ABB RobotStudio station: ScenarioBrakeTest.rspag

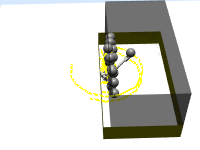
--- station ---
Station Solution10_1 (saved by RobotStudio 6.7.7850.130)
Controller IRB_6700_175kg_3.05m
  mechanical unit ROB_1: IRB6700_175_305__04, 6 joints, base frame (0, 0, 0) mm
Layout (positions relative to the parent item):
  - IRB6700_175_305__04 [mechanism, from Robots\IRB6700_175_305__04.rslib] at (0, 0, 0) mm; joint values [-1.1842, -1.1345, -1.3411, 0, 0.5236, 0] (rad or m)
  - MyNewTool [mechanism] at (-813.86, 1999.53, 2271.97) mm, rotated rx 0 ry -21.84 rz -67.85 deg
      TCP MyNewTool at (0, 0, 0) mm
      links: IsoPlate_large_sat
  - SafeSpaceGeometries [graphiccomponentgroup]
    - safety zone [part]
    - tcp blob [part] at (-813.86, 1999.53, 2271.97) mm, rotated rx 0 ry -21.84 rz -67.85 deg
    - tcp blob [part] at (-1295.95, 228.51, 2690.77) mm, rotated rx -180 ry 87.5 rz -10 deg
    - tcp blob [part] at (-2238.8, 394.76, 1689.63) mm, rotated rx -180 ry 50 rz -10 deg
    - tcp blob [part] at (2430.82, 428.62, 1082.75) mm, rotated rx 0 ry -62.5 rz -170 deg
    - tcp blob [part] at (2269.78, 400.22, 2021.28) mm, rotated rx 0 ry -31.25 rz -170 deg
    - tcp blob [part] at (1652.62, 291.4, 2738.82) mm, rotated rx 0 ry 0 rz -170 deg
    - tcp blob [part] at (758.42, 133.73, 3027.14) mm, rotated rx 0 ry 31.25 rz -170 deg
    - tcp blob [part] at (1942.58, 342.53, 1802.45) mm, rotated rx 0 ry -56.25 rz -170 deg
    - tcp blob [part] at (1681.88, 296.56, 2717.61) mm, rotated rx 0 ry -25 rz -170 deg
    - tcp blob [part] at (991.45, 174.82, 3362.65) mm, rotated rx 0 ry 6.25 rz -170 deg
    - tcp blob [part] at (863.06, 152.18, 2986.78) mm, rotated rx 0 ry -18.75 rz -170 deg
    - tcp blob [part] at (582.02, 504.32, 3027.14) mm, rotated rx 0 ry 31.25 rz -139.09 deg
    - tcp blob [part] at (82.99, 71.91, 2781.05) mm, rotated rx 0 ry -12.5 rz -139.09 deg
    - tcp blob [part] at (34.09, 103.78, 3551.67) mm, rotated rx 0 ry 12.5 rz -108.18 deg
    - tcp blob [part] at (34.26, 104.33, 2781.05) mm, rotated rx 0 ry -12.5 rz -108.18 deg
    - tcp blob [part] at (-24.07, 106.55, 3551.67) mm, rotated rx 0 ry 12.5 rz -77.27 deg
    - tcp blob [part] at (-24.19, 107.11, 2781.05) mm, rotated rx 0 ry -12.5 rz -77.27 deg
    - tcp blob [part] at (-531.44, 557.36, 3027.14) mm, rotated rx 0 ry 31.25 rz -46.36 deg
    - tcp blob [part] at (-75.78, 79.47, 2781.05) mm, rotated rx 0 ry -12.5 rz -46.36 deg
    - tcp blob [part] at (-1617.44, 447.17, 2738.82) mm, rotated rx 0 ry 0 rz -15.45 deg
    - tcp blob [part] at (-742.27, 205.22, 3027.14) mm, rotated rx 0 ry 31.25 rz -15.45 deg
    - tcp blob [part] at (-970.35, 268.27, 3362.65) mm, rotated rx 0 ry 6.25 rz -15.45 deg
    - tcp blob [part] at (-844.68, 233.53, 2986.78) mm, rotated rx 0 ry -18.75 rz -15.45 deg
    - tcp blob [part] at (1020.75, 282.21, 1205.4) mm, rotated rx -180 ry 55 rz -164.55 deg
    - tcp blob [part] at (1369.56, 378.64, 2484.63) mm, rotated rx -180 ry 80 rz -164.55 deg
    - tcp blob [part] at (1491.26, 412.29, 1540.36) mm, rotated rx -180 ry 48.75 rz -164.55 deg
    - tcp blob [part] at (1123.15, 310.52, 667.59) mm, rotated rx -180 ry 17.5 rz -164.55 deg
    - tcp blob [part] at (-1042.95, 183.9, 1205.4) mm, rotated rx -180 ry 55 rz -10 deg
    - tcp blob [part] at (-1399.35, 246.74, 2484.63) mm, rotated rx -180 ry 80 rz -10 deg
    - tcp blob [part] at (-1523.7, 268.67, 1540.36) mm, rotated rx -180 ry 48.75 rz -10 deg
    - tcp blob [part] at (-1147.59, 202.35, 667.59) mm, rotated rx -180 ry 17.5 rz -10 deg
    - tcp blob [part] at (-1669.17, 294.32, 3217.01) mm, rotated rx 0 ry 75 rz 170 deg
    - tcp blob [part] at (-2174.87, 383.49, 2414.57) mm, rotated rx -180 ry 73.75 rz -10 deg
    - tcp blob [part] at (-2197.25, 387.43, 1462.17) mm, rotated rx -180 ry 42.5 rz -10 deg
    - tcp blob [part] at (-1729.8, 305.01, 636.16) mm, rotated rx -180 ry 11.25 rz -10 deg
    - tcp blob [part] at (-1641.43, 289.43, 3240.22) mm, rotated rx 0 ry 50 rz 170 deg
    - tcp blob [part] at (-2433.72, 429.13, 2729.98) mm, rotated rx 0 ry 81.25 rz 170 deg
    - tcp blob [part] at (-2109.4, 371.94, 2506.76) mm, rotated rx 0 ry 56.25 rz 170 deg
    - fence_2000 [part]
    - fence_4000 [part]
    - fence_6000 [part]
  - Part_2 [part] at (-12128.6, -11086.49, -16.13) mm
Attachment: MyNewTool is attached to IRB6700_175_305__04 / Link6
Attachment: tcp blob is attached to IRB6700_175_305__04 / Link6
Collision set zone collisions: tcp blob against safety zone, near miss 0 m
Targets, tools, work objects and paths stored in the station and not in the controller backup, written as RAPID:
! task T_ROB1
MODULE Module1
  CONST robtarget Target_0112:=[[2430.822564059,428.619603359,1082.747931027],[0.074510479,-0.516799169,-0.045214069,-0.851658673],[-2,0,0,6],[9E+09,9E+09,9E+09,9E+09,9E+09,9E+09]];
  CONST robtarget Target_0113:=[[2430.822564059,428.619603359,1082.747931027],[0.074510479,-0.516799169,-0.045214069,-0.851658673],[-2,0,0,6],[9E+09,9E+09,9E+09,9E+09,9E+09,9E+09]];
  CONST robtarget Target_0114:=[[2269.784024949,400.22416398,2021.283364573],[0.083934914,-0.268315134,-0.023474532,-0.959380459],[-2,0,0,6],[9E+09,9E+09,9E+09,9E+09,9E+09,9E+09]];
  CONST robtarget Target_0115:=[[2269.784024949,400.22416398,2021.283364573],[0.083934914,-0.268315134,-0.023474532,-0.959380459],[-2,0,0,6],[9E+09,9E+09,9E+09,9E+09,9E+09,9E+09]];
  CONST robtarget Target_0116:=[[1652.620090316,291.401510784,2738.817182602],[0.087155743,0,0,-0.996194698],[-2,0,0,4],[9E+09,9E+09,9E+09,9E+09,9E+09,9E+09]];
  CONST robtarget Target_0117:=[[1652.620090316,291.401510784,2738.817182602],[0.087155743,0,0,-0.996194698],[-2,0,0,4],[9E+09,9E+09,9E+09,9E+09,9E+09,9E+09]];
  CONST robtarget Target_0118:=[[758.417081686,133.729394131,3027.138106342],[0.083934914,0.268315134,0.023474532,-0.959380459],[-2,0,0,4],[9E+09,9E+09,9E+09,9E+09,9E+09,9E+09]];
  CONST robtarget Target_0119:=[[758.417081686,133.729394131,3027.138106342],[0.083934914,0.268315134,0.023474532,-0.959380459],[-2,0,0,4],[9E+09,9E+09,9E+09,9E+09,9E+09,9E+09]];
  CONST robtarget Target_0120:=[[1942.582099481,342.52963638,1802.454040912],[0.076864503,-0.46960293,-0.041084933,-0.878565288],[-2,0,0,6],[9E+09,9E+09,9E+09,9E+09,9E+09,9E+09]];
  CONST robtarget Target_0121:=[[1942.582099481,342.52963638,1802.454040912],[0.076864503,-0.46960293,-0.041084933,-0.878565288],[-2,0,0,6],[9E+09,9E+09,9E+09,9E+09,9E+09,9E+09]];
  CONST robtarget Target_0122:=[[1681.877573603,296.560394475,2717.608919096],[0.085089804,-0.215615996,-0.018863955,-0.972580906],[-2,0,0,6],[9E+09,9E+09,9E+09,9E+09,9E+09,9E+09]];
  CONST robtarget Target_0123:=[[1681.877573603,296.560394475,2717.608919096],[0.085089804,-0.215615996,-0.018863955,-0.972580906],[-2,0,0,6],[9E+09,9E+09,9E+09,9E+09,9E+09,9E+09]];
  CONST robtarget Target_0124:=[[991.452940755,174.819903558,3362.652755828],[0.08702614,0.054307058,0.004751252,-0.994713336],[-2,0,0,6],[9E+09,9E+09,9E+09,9E+09,9E+09,9E+09]];
  CONST robtarget Target_0125:=[[991.452940755,174.819903558,3362.652755828],[0.08702614,0.054307058,0.004751252,-0.994713336],[-2,0,0,6],[9E+09,9E+09,9E+09,9E+09,9E+09,9E+09]];
  CONST robtarget Target_0126:=[[863.057219085,152.18027362,2986.783074619],[0.085991632,-0.162275607,-0.014197276,-0.982888856],[-2,0,0,6],[9E+09,9E+09,9E+09,9E+09,9E+09,9E+09]];
  CONST robtarget Target_0127:=[[863.057219085,152.18027362,2986.783074619],[0.085991632,-0.162275607,-0.014197276,-0.982888856],[-2,0,0,6],[9E+09,9E+09,9E+09,9E+09,9E+09,9E+09]];
  CONST robtarget Target_0128:=[[582.015510048,504.319310271,3027.138106342],[0.336549779,0.252358089,0.094124701,-0.902324876],[-2,0,0,4],[9E+09,9E+09,9E+09,9E+09,9E+09,9E+09]];
  CONST robtarget Target_0129:=[[582.015510048,504.319310271,3027.138106342],[0.336549779,0.252358089,0.094124701,-0.902324876],[-2,0,0,4],[9E+09,9E+09,9E+09,9E+09,9E+09,9E+09]];
  CONST robtarget Target_0130:=[[-531.441500554,557.359804917,3027.138106342],[0.885289165,0.106025771,0.24759362,-0.379102928],[-1,0,0,4],[9E+09,9E+09,9E+09,9E+09,9E+09,9E+09]];
  CONST robtarget Target_0131:=[[-531.441500554,557.359804917,3027.138106342],[0.885289165,0.106025771,0.24759362,-0.379102928],[-1,0,0,4],[9E+09,9E+09,9E+09,9E+09,9E+09,9E+09]];
  CONST robtarget Target_0132:=[[-1617.437423958,447.173549064,2738.817182602],[0.99091931,0,0,-0.134457877],[-1,0,0,4],[9E+09,9E+09,9E+09,9E+09,9E+09,9E+09]];
  CONST robtarget Target_0133:=[[-742.271123337,205.215984046,3027.138106342],[0.954300023,0.036214892,0.26689426,-0.129489005],[-1,0,0,4],[9E+09,9E+09,9E+09,9E+09,9E+09,9E+09]];
  CONST robtarget Target_0134:=[[-742.271123337,205.215984046,3027.138106342],[0.954300023,0.036214892,0.26689426,-0.129489005],[-1,0,0,4],[9E+09,9E+09,9E+09,9E+09,9E+09,9E+09]];
  CONST robtarget Target_0135:=[[-970.345876749,268.271899177,3362.652755828],[0.989445792,0.007329904,0.054019472,-0.134257935],[-1,0,0,6],[9E+09,9E+09,9E+09,9E+09,9E+09,9E+09]];
  CONST robtarget Target_0136:=[[-970.345876749,268.271899177,3362.652755828],[0.989445792,0.007329904,0.054019472,-0.134257935],[-1,0,0,6],[9E+09,9E+09,9E+09,9E+09,9E+09,9E+09]];
  CONST robtarget Target_0137:=[[-844.683574492,233.529993956,2986.783074619],[0.97768393,-0.02190258,-0.16141627,-0.132661968],[-1,0,0,6],[9E+09,9E+09,9E+09,9E+09,9E+09,9E+09]];
  CONST robtarget Target_0138:=[[-844.683574492,233.529993956,2986.783074619],[0.97768393,-0.02190258,-0.16141627,-0.132661968],[-1,0,0,6],[9E+09,9E+09,9E+09,9E+09,9E+09,9E+09]];
  CONST robtarget Target_0139:=[[1020.749593142,282.207034108,1205.399859098],[0.457555617,-0.119265594,0.878956163,0.062085738],[0,0,0,0],[9E+09,9E+09,9E+09,9E+09,9E+09,9E+09]];
  CONST robtarget Target_0140:=[[1369.555461946,378.641527324,2484.633262527],[0.636950655,-0.10300071,0.759088231,0.086427857],[0,0,0,0],[9E+09,9E+09,9E+09,9E+09,9E+09,9E+09]];
  CONST robtarget Target_0141:=[[1491.258427618,412.28879323,1540.363850907],[0.408959365,-0.122472816,0.902592553,0.055491711],[0,0,0,0],[9E+09,9E+09,9E+09,9E+09,9E+09,9E+09]];
  CONST robtarget Target_0142:=[[1123.154360792,310.518919757,667.591967242],[0.150742001,-0.132892991,0.979386506,0.020454188],[0,0,0,0],[9E+09,9E+09,9E+09,9E+09,9E+09,9E+09]];
  CONST robtarget Target_0143:=[[2430.822564059,428.619603359,1082.747931027],[0.074510479,-0.516799169,-0.045214069,-0.851658673],[-2,0,0,6],[9E+09,9E+09,9E+09,9E+09,9E+09,9E+09]];
  CONST robtarget Target_0144:=[[2430.822564059,428.619603359,1082.747931027],[0.074510479,-0.516799169,-0.045214069,-0.851658673],[-2,0,0,6],[9E+09,9E+09,9E+09,9E+09,9E+09,9E+09]];
  CONST robtarget Target_0145:=[[2269.784024949,400.22416398,2021.283364573],[0.083934914,-0.268315134,-0.023474532,-0.959380459],[-2,0,0,6],[9E+09,9E+09,9E+09,9E+09,9E+09,9E+09]];
  CONST robtarget Target_0146:=[[2269.784024949,400.22416398,2021.283364573],[0.083934914,-0.268315134,-0.023474532,-0.959380459],[-2,0,0,6],[9E+09,9E+09,9E+09,9E+09,9E+09,9E+09]];
  CONST robtarget Target_0147:=[[1652.620090316,291.401510784,2738.817182602],[0.087155743,0,0,-0.996194698],[-2,0,0,4],[9E+09,9E+09,9E+09,9E+09,9E+09,9E+09]];
  CONST robtarget Target_0148:=[[1652.620090316,291.401510784,2738.817182602],[0.087155743,0,0,-0.996194698],[-2,0,0,4],[9E+09,9E+09,9E+09,9E+09,9E+09,9E+09]];
  CONST robtarget Target_0149:=[[758.417081686,133.729394131,3027.138106342],[0.083934914,0.268315134,0.023474532,-0.959380459],[-2,0,0,4],[9E+09,9E+09,9E+09,9E+09,9E+09,9E+09]];
  CONST robtarget Target_0150:=[[758.417081686,133.729394131,3027.138106342],[0.083934914,0.268315134,0.023474532,-0.959380459],[-2,0,0,4],[9E+09,9E+09,9E+09,9E+09,9E+09,9E+09]];
  CONST robtarget Target_0151:=[[1942.582099481,342.52963638,1802.454040912],[0.076864503,-0.46960293,-0.041084933,-0.878565288],[-2,0,0,6],[9E+09,9E+09,9E+09,9E+09,9E+09,9E+09]];
  CONST robtarget Target_0152:=[[1942.582099481,342.52963638,1802.454040912],[0.076864503,-0.46960293,-0.041084933,-0.878565288],[-2,0,0,6],[9E+09,9E+09,9E+09,9E+09,9E+09,9E+09]];
  CONST robtarget Target_0153:=[[1681.877573603,296.560394475,2717.608919096],[0.085089804,-0.215615996,-0.018863955,-0.972580906],[-2,0,0,6],[9E+09,9E+09,9E+09,9E+09,9E+09,9E+09]];
  CONST robtarget Target_0154:=[[1681.877573603,296.560394475,2717.608919096],[0.085089804,-0.215615996,-0.018863955,-0.972580906],[-2,0,0,6],[9E+09,9E+09,9E+09,9E+09,9E+09,9E+09]];
  CONST robtarget Target_0155:=[[991.452940755,174.819903558,3362.652755828],[0.08702614,0.054307058,0.004751252,-0.994713336],[-2,0,0,6],[9E+09,9E+09,9E+09,9E+09,9E+09,9E+09]];
  CONST robtarget Target_0156:=[[991.452940755,174.819903558,3362.652755828],[0.08702614,0.054307058,0.004751252,-0.994713336],[-2,0,0,6],[9E+09,9E+09,9E+09,9E+09,9E+09,9E+09]];
  CONST robtarget Target_0157:=[[863.057219085,152.18027362,2986.783074619],[0.085991632,-0.162275607,-0.014197276,-0.982888856],[-2,0,0,6],[9E+09,9E+09,9E+09,9E+09,9E+09,9E+09]];
  CONST robtarget Target_0158:=[[863.057219085,152.18027362,2986.783074619],[0.085991632,-0.162275607,-0.014197276,-0.982888856],[-2,0,0,6],[9E+09,9E+09,9E+09,9E+09,9E+09,9E+09]];
  CONST robtarget Target_0159:=[[582.015510048,504.319310271,3027.138106342],[0.336549779,0.252358089,0.094124701,-0.902324876],[-2,0,0,4],[9E+09,9E+09,9E+09,9E+09,9E+09,9E+09]];
  CONST robtarget Target_0160:=[[582.015510048,504.319310271,3027.138106342],[0.336549779,0.252358089,0.094124701,-0.902324876],[-2,0,0,4],[9E+09,9E+09,9E+09,9E+09,9E+09,9E+09]];
  CONST robtarget Target_0161:=[[-531.441500554,557.359804917,3027.138106342],[0.885289165,0.106025771,0.24759362,-0.379102928],[-1,0,0,4],[9E+09,9E+09,9E+09,9E+09,9E+09,9E+09]];
  CONST robtarget Target_0162:=[[-531.441500554,557.359804917,3027.138106342],[0.885289165,0.106025771,0.24759362,-0.379102928],[-1,0,0,4],[9E+09,9E+09,9E+09,9E+09,9E+09,9E+09]];
  CONST robtarget Target_0163:=[[-1617.437423958,447.173549064,2738.817182602],[0.99091931,0,0,-0.134457877],[-1,0,0,4],[9E+09,9E+09,9E+09,9E+09,9E+09,9E+09]];
  CONST robtarget Target_0164:=[[-742.271123337,205.215984046,3027.138106342],[0.954300023,0.036214892,0.26689426,-0.129489005],[-1,0,0,4],[9E+09,9E+09,9E+09,9E+09,9E+09,9E+09]];
  CONST robtarget Target_0165:=[[-742.271123337,205.215984046,3027.138106342],[0.954300023,0.036214892,0.26689426,-0.129489005],[-1,0,0,4],[9E+09,9E+09,9E+09,9E+09,9E+09,9E+09]];
  CONST robtarget Target_0166:=[[-970.345876749,268.271899177,3362.652755828],[0.989445792,0.007329904,0.054019472,-0.134257935],[-1,0,0,6],[9E+09,9E+09,9E+09,9E+09,9E+09,9E+09]];
  CONST robtarget Target_0167:=[[-970.345876749,268.271899177,3362.652755828],[0.989445792,0.007329904,0.054019472,-0.134257935],[-1,0,0,6],[9E+09,9E+09,9E+09,9E+09,9E+09,9E+09]];
  CONST robtarget Target_0168:=[[-844.683574492,233.529993956,2986.783074619],[0.97768393,-0.02190258,-0.16141627,-0.132661968],[-1,0,0,6],[9E+09,9E+09,9E+09,9E+09,9E+09,9E+09]];
  CONST robtarget Target_0169:=[[-844.683574492,233.529993956,2986.783074619],[0.97768393,-0.02190258,-0.16141627,-0.132661968],[-1,0,0,6],[9E+09,9E+09,9E+09,9E+09,9E+09,9E+09]];
  CONST robtarget Target_0170:=[[1020.749593142,282.207034108,1205.399859098],[0.457555617,-0.119265594,0.878956163,0.062085738],[0,0,0,0],[9E+09,9E+09,9E+09,9E+09,9E+09,9E+09]];
  CONST robtarget Target_0171:=[[1369.555461946,378.641527324,2484.633262527],[0.636950655,-0.10300071,0.759088231,0.086427857],[0,0,0,0],[9E+09,9E+09,9E+09,9E+09,9E+09,9E+09]];
  CONST robtarget Target_0172:=[[1491.258427618,412.28879323,1540.363850907],[0.408959365,-0.122472816,0.902592553,0.055491711],[0,0,0,0],[9E+09,9E+09,9E+09,9E+09,9E+09,9E+09]];
  CONST robtarget Target_0173:=[[1123.154360792,310.518919757,667.591967242],[0.150742001,-0.132892991,0.979386506,0.020454188],[0,0,0,0],[9E+09,9E+09,9E+09,9E+09,9E+09,9E+09]];
  CONST robtarget Target_0174:=[[2430.822564059,428.619603359,1082.747931027],[0.074510479,-0.516799169,-0.045214069,-0.851658673],[-2,0,0,6],[9E+09,9E+09,9E+09,9E+09,9E+09,9E+09]];
  CONST robtarget Target_0175:=[[2430.822564059,428.619603359,1082.747931027],[0.074510479,-0.516799169,-0.045214069,-0.851658673],[-2,0,0,6],[9E+09,9E+09,9E+09,9E+09,9E+09,9E+09]];
  CONST robtarget Target_0176:=[[2269.784024949,400.22416398,2021.283364573],[0.083934914,-0.268315134,-0.023474532,-0.959380459],[-2,0,0,6],[9E+09,9E+09,9E+09,9E+09,9E+09,9E+09]];
  CONST robtarget Target_0177:=[[2269.784024949,400.22416398,2021.283364573],[0.083934914,-0.268315134,-0.023474532,-0.959380459],[-2,0,0,6],[9E+09,9E+09,9E+09,9E+09,9E+09,9E+09]];
  CONST robtarget Target_0178:=[[1652.620090316,291.401510784,2738.817182602],[0.087155743,0,0,-0.996194698],[-2,0,0,4],[9E+09,9E+09,9E+09,9E+09,9E+09,9E+09]];
  CONST robtarget Target_0179:=[[1652.620090316,291.401510784,2738.817182602],[0.087155743,0,0,-0.996194698],[-2,0,0,4],[9E+09,9E+09,9E+09,9E+09,9E+09,9E+09]];
  CONST robtarget Target_0180:=[[758.417081686,133.729394131,3027.138106342],[0.083934914,0.268315134,0.023474532,-0.959380459],[-2,0,0,4],[9E+09,9E+09,9E+09,9E+09,9E+09,9E+09]];
  CONST robtarget Target_0181:=[[758.417081686,133.729394131,3027.138106342],[0.083934914,0.268315134,0.023474532,-0.959380459],[-2,0,0,4],[9E+09,9E+09,9E+09,9E+09,9E+09,9E+09]];
  CONST robtarget Target_0182:=[[1942.582099481,342.52963638,1802.454040912],[0.076864503,-0.46960293,-0.041084933,-0.878565288],[-2,0,0,6],[9E+09,9E+09,9E+09,9E+09,9E+09,9E+09]];
  CONST robtarget Target_0183:=[[1942.582099481,342.52963638,1802.454040912],[0.076864503,-0.46960293,-0.041084933,-0.878565288],[-2,0,0,6],[9E+09,9E+09,9E+09,9E+09,9E+09,9E+09]];
  CONST robtarget Target_0184:=[[1681.877573603,296.560394475,2717.608919096],[0.085089804,-0.215615996,-0.018863955,-0.972580906],[-2,0,0,6],[9E+09,9E+09,9E+09,9E+09,9E+09,9E+09]];
  CONST robtarget Target_0185:=[[1681.877573603,296.560394475,2717.608919096],[0.085089804,-0.215615996,-0.018863955,-0.972580906],[-2,0,0,6],[9E+09,9E+09,9E+09,9E+09,9E+09,9E+09]];
  CONST robtarget Target_0186:=[[991.452940755,174.819903558,3362.652755828],[0.08702614,0.054307058,0.004751252,-0.994713336],[-2,0,0,6],[9E+09,9E+09,9E+09,9E+09,9E+09,9E+09]];
  CONST robtarget Target_0187:=[[991.452940755,174.819903558,3362.652755828],[0.08702614,0.054307058,0.004751252,-0.994713336],[-2,0,0,6],[9E+09,9E+09,9E+09,9E+09,9E+09,9E+09]];
  CONST robtarget Target_0188:=[[863.057219085,152.18027362,2986.783074619],[0.085991632,-0.162275607,-0.014197276,-0.982888856],[-2,0,0,6],[9E+09,9E+09,9E+09,9E+09,9E+09,9E+09]];
  CONST robtarget Target_0189:=[[863.057219085,152.18027362,2986.783074619],[0.085991632,-0.162275607,-0.014197276,-0.982888856],[-2,0,0,6],[9E+09,9E+09,9E+09,9E+09,9E+09,9E+09]];
  CONST robtarget Target_0190:=[[582.015510048,504.319310271,3027.138106342],[0.336549779,0.252358089,0.094124701,-0.902324876],[-2,0,0,4],[9E+09,9E+09,9E+09,9E+09,9E+09,9E+09]];
  CONST robtarget Target_0191:=[[582.015510048,504.319310271,3027.138106342],[0.336549779,0.252358089,0.094124701,-0.902324876],[-2,0,0,4],[9E+09,9E+09,9E+09,9E+09,9E+09,9E+09]];
  CONST robtarget Target_0192:=[[-531.441500554,557.359804917,3027.138106342],[0.885289165,0.106025771,0.24759362,-0.379102928],[-1,0,0,4],[9E+09,9E+09,9E+09,9E+09,9E+09,9E+09]];
  CONST robtarget Target_0193:=[[-531.441500554,557.359804917,3027.138106342],[0.885289165,0.106025771,0.24759362,-0.379102928],[-1,0,0,4],[9E+09,9E+09,9E+09,9E+09,9E+09,9E+09]];
  CONST robtarget Target_0194:=[[-1617.437423958,447.173549064,2738.817182602],[0.99091931,0,0,-0.134457877],[-1,0,0,4],[9E+09,9E+09,9E+09,9E+09,9E+09,9E+09]];
  CONST robtarget Target_0195:=[[-742.271123337,205.215984046,3027.138106342],[0.954300023,0.036214892,0.26689426,-0.129489005],[-1,0,0,4],[9E+09,9E+09,9E+09,9E+09,9E+09,9E+09]];
  CONST robtarget Target_0196:=[[-742.271123337,205.215984046,3027.138106342],[0.954300023,0.036214892,0.26689426,-0.129489005],[-1,0,0,4],[9E+09,9E+09,9E+09,9E+09,9E+09,9E+09]];
  CONST robtarget Target_0197:=[[-970.345876749,268.271899177,3362.652755828],[0.989445792,0.007329904,0.054019472,-0.134257935],[-1,0,0,6],[9E+09,9E+09,9E+09,9E+09,9E+09,9E+09]];
  CONST robtarget Target_0198:=[[-970.345876749,268.271899177,3362.652755828],[0.989445792,0.007329904,0.054019472,-0.134257935],[-1,0,0,6],[9E+09,9E+09,9E+09,9E+09,9E+09,9E+09]];
  CONST robtarget Target_0199:=[[-844.683574492,233.529993956,2986.783074619],[0.97768393,-0.02190258,-0.16141627,-0.132661968],[-1,0,0,6],[9E+09,9E+09,9E+09,9E+09,9E+09,9E+09]];
  CONST robtarget Target_0200:=[[-844.683574492,233.529993956,2986.783074619],[0.97768393,-0.02190258,-0.16141627,-0.132661968],[-1,0,0,6],[9E+09,9E+09,9E+09,9E+09,9E+09,9E+09]];
  CONST robtarget Target_0201:=[[1020.749593142,282.207034108,1205.399859098],[0.457555617,-0.119265594,0.878956163,0.062085738],[0,0,0,0],[9E+09,9E+09,9E+09,9E+09,9E+09,9E+09]];
  CONST robtarget Target_0202:=[[1369.555461946,378.641527324,2484.633262527],[0.636950655,-0.10300071,0.759088231,0.086427857],[0,0,0,0],[9E+09,9E+09,9E+09,9E+09,9E+09,9E+09]];
  CONST robtarget Target_0203:=[[1491.258427618,412.28879323,1540.363850907],[0.408959365,-0.122472816,0.902592553,0.055491711],[0,0,0,0],[9E+09,9E+09,9E+09,9E+09,9E+09,9E+09]];
  CONST robtarget Target_0204:=[[1123.154360792,310.518919757,667.591967242],[0.150742001,-0.132892991,0.979386506,0.020454188],[0,0,0,0],[9E+09,9E+09,9E+09,9E+09,9E+09,9E+09]];
ENDMODULE


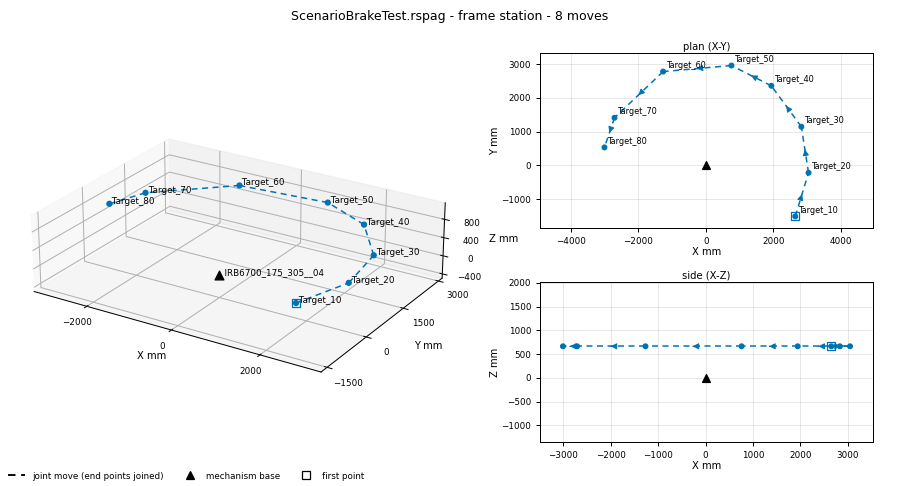
[picture p0: tool path of ScenarioBrakeTest.rspag in frame station, 8 of 130 moves have a stored position in this frame; points joined in program order, loops and branches not executed]
--- Backups/IRB_6700_175kg_3.05m/RAPID/TASK1/PROGMOD/CalibData.mod ---
MODULE CalibData
	PERS tooldata MyNewTool:=[TRUE,[[0,0,0],[1,0,0,0]],[175,[0,0,1],[1,0,0,0],17.5,17.5,17.5]];
ENDMODULE

--- Backups/IRB_6700_175kg_3.05m/RAPID/TASK1/PROGMOD/Module1.mod ---
MODULE Module1
	CONST robtarget Target_10:=[[2650.778985035,-1514.394022891,665.53670734],[0.237207259,0.063532185,0.962557826,-0.114798994],[-1,0,-1,0],[9E+09,9E+09,9E+09,9E+09,9E+09,9E+09]];
	CONST robtarget Target_20:=[[3044.708925288,-223.083043607,665.53670734],[0.256719524,-0.150874772,0.952780515,-0.059507803],[-1,0,-1,0],[9E+09,9E+09,9E+09,9E+09,9E+09,9E+09]];
	CONST robtarget Target_30:=[[2830.995781706,1142.576635519,665.53670734],[0.263526219,-0.362657835,0.893886571,0.000156031],[0,0,-1,0],[9E+09,9E+09,9E+09,9E+09,9E+09,9E+09]];
	CONST robtarget Target_40:=[[1941.519398723,2355.954351946,665.53670734],[0.255362535,-0.571733158,0.776965317,0.065085085],[0,0,-1,0],[9E+09,9E+09,9E+09,9E+09,9E+09,9E+09]];
	CONST robtarget Target_50:=[[758.480316395,2957.148304315,665.53670734],[0.235112529,-0.726933226,0.634130896,0.119030212],[0,0,-1,0],[9E+09,9E+09,9E+09,9E+09,9E+09,9E+09]];
	CONST robtarget Target_60:=[[-1267.010409106,2777.53543763,665.53670734],[0.182049336,-0.896624462,0.355834908,0.190536432],[1,0,-1,0],[9E+09,9E+09,9E+09,9E+09,9E+09,9E+09]];
	CONST robtarget Target_70:=[[-2708.612226105,1408.345942114,665.53670734],[0.110083745,-0.963626329,0.044477023,0.239431956],[1,0,-1,0],[9E+09,9E+09,9E+09,9E+09,9E+09,9E+09]];
	CONST robtarget Target_80:=[[-3006.534548987,529.875919266,665.53670734],[0.072430236,-0.959197766,-0.102438045,0.253377098],[1,0,-1,0],[9E+09,9E+09,9E+09,9E+09,9E+09,9E+09]];
	CONST jointtarget JointTarget_1:=[[170.000007007,85,-98.742260129,0.112841515,40.027258121,-22.258237543],[9E+09,9E+09,9E+09,9E+09,9E+09,9E+09]];
	CONST jointtarget JointTarget_2:=[[143.024262269,85,-98.742260129,0.112841515,40.027258121,-22.258237543],[9E+09,9E+09,9E+09,9E+09,9E+09,9E+09]];
	CONST jointtarget JointTarget_3:=[[113.3049809,85,-98.742260129,0.112841515,40.027258121,-22.258237543],[9E+09,9E+09,9E+09,9E+09,9E+09,9E+09]];
	CONST jointtarget JointTarget_4:=[[87.274335878,85,-98.742260129,0.112841515,40.027258121,-22.258237543],[9E+09,9E+09,9E+09,9E+09,9E+09,9E+09]];
	CONST jointtarget JointTarget_5:=[[48.429291781,85,-98.742260129,0.112841515,40.027258121,-22.258237543],[9E+09,9E+09,9E+09,9E+09,9E+09,9E+09]];
	CONST jointtarget JointTarget_6:=[[15.425917994,85,-98.742260129,0.112841515,40.027258121,-22.258237543],[9E+09,9E+09,9E+09,9E+09,9E+09,9E+09]];
	CONST jointtarget JointTarget_7:=[[-5.037431675,85,-98.742260129,0.112841515,40.027258121,-22.258237543],[9E+09,9E+09,9E+09,9E+09,9E+09,9E+09]];
	CONST jointtarget JointTarget_8:=[[-30.266766578,85,-98.742260129,0.112841515,40.027258121,-22.258237543],[9E+09,9E+09,9E+09,9E+09,9E+09,9E+09]];
	CONST jointtarget JointTarget_9:=[[-58.818282132,85,-98.742260129,0.112841515,40.027258121,-22.258237543],[9E+09,9E+09,9E+09,9E+09,9E+09,9E+09]];
	CONST jointtarget JointTarget_10:=[[-77.492415908,85,-98.742260129,0.112841515,40.027258121,-22.258237543],[9E+09,9E+09,9E+09,9E+09,9E+09,9E+09]];
	CONST jointtarget JointTarget_11:=[[-105.198837588,85,-98.742260129,0.112841515,40.027258121,-22.258237543],[9E+09,9E+09,9E+09,9E+09,9E+09,9E+09]];
	CONST jointtarget Target_02:=[[227.295779513,-27.5,0,0,30,0],[9E+09,9E+09,9E+09,9E+09,9E+09,9E+09]];
	CONST jointtarget Target_01:=[[170,-27.5,0,0,30,0],[9E+09,9E+09,9E+09,9E+09,9E+09,9E+09]];
	CONST jointtarget Target_03:=[[284.591559026,-27.5,0,0,30,0],[9E+09,9E+09,9E+09,9E+09,9E+09,9E+09]];
	CONST jointtarget Target_05:=[[227.295779513,10,0,0,30,0],[9E+09,9E+09,9E+09,9E+09,9E+09,9E+09]];
	CONST jointtarget Target_04:=[[170,10,0,0,30,0],[9E+09,9E+09,9E+09,9E+09,9E+09,9E+09]];
	CONST jointtarget Target_06:=[[284.591559026,10,0,0,30,0],[9E+09,9E+09,9E+09,9E+09,9E+09,9E+09]];
	CONST jointtarget Target_08:=[[-170,-65,-117.5,0,30,0],[9E+09,9E+09,9E+09,9E+09,9E+09,9E+09]];
	CONST jointtarget Target_07:=[[-170,-65,-117.5,0,30,0],[9E+09,9E+09,9E+09,9E+09,9E+09,9E+09]];
	CONST jointtarget Target_09:=[[164.374588252,-65,-117.5,0,30,0],[9E+09,9E+09,9E+09,9E+09,9E+09,9E+09]];
	CONST jointtarget Target_011:=[[-170,-65,-86.25,0,30,0],[9E+09,9E+09,9E+09,9E+09,9E+09,9E+09]];
	CONST jointtarget Target_010:=[[-170,-65,-86.25,0,30,0],[9E+09,9E+09,9E+09,9E+09,9E+09,9E+09]];
	CONST jointtarget Target_012:=[[164.374588252,-65,-86.25,0,30,0],[9E+09,9E+09,9E+09,9E+09,9E+09,9E+09]];
	CONST jointtarget Target_014:=[[-170,-65,-55,0,30,0],[9E+09,9E+09,9E+09,9E+09,9E+09,9E+09]];
	CONST jointtarget Target_013:=[[-170,-65,-55,0,30,0],[9E+09,9E+09,9E+09,9E+09,9E+09,9E+09]];
	CONST jointtarget Target_015:=[[164.374588252,-65,-55,0,30,0],[9E+09,9E+09,9E+09,9E+09,9E+09,9E+09]];
	CONST jointtarget Target_017:=[[-170,-65,-23.75,0,30,0],[9E+09,9E+09,9E+09,9E+09,9E+09,9E+09]];
	CONST jointtarget Target_016:=[[-170,-65,-23.75,0,30,0],[9E+09,9E+09,9E+09,9E+09,9E+09,9E+09]];
	CONST jointtarget Target_018:=[[164.374588252,-65,-23.75,0,30,0],[9E+09,9E+09,9E+09,9E+09,9E+09,9E+09]];
	CONST jointtarget Target_020:=[[-170,-27.5,-148.75,0,30,0],[9E+09,9E+09,9E+09,9E+09,9E+09,9E+09]];
	CONST jointtarget Target_019:=[[-170,-27.5,-148.75,0,30,0],[9E+09,9E+09,9E+09,9E+09,9E+09,9E+09]];
	CONST jointtarget Target_021:=[[164.374588252,-27.5,-148.75,0,30,0],[9E+09,9E+09,9E+09,9E+09,9E+09,9E+09]];
	CONST jointtarget Target_023:=[[-170,-27.5,-117.5,0,30,0],[9E+09,9E+09,9E+09,9E+09,9E+09,9E+09]];
	CONST jointtarget Target_022:=[[-170,-27.5,-117.5,0,30,0],[9E+09,9E+09,9E+09,9E+09,9E+09,9E+09]];
	CONST jointtarget Target_024:=[[164.374588252,-27.5,-117.5,0,30,0],[9E+09,9E+09,9E+09,9E+09,9E+09,9E+09]];
	CONST jointtarget Target_026:=[[-170,-27.5,-86.25,0,30,0],[9E+09,9E+09,9E+09,9E+09,9E+09,9E+09]];
	CONST jointtarget Target_025:=[[-170,-27.5,-86.25,0,30,0],[9E+09,9E+09,9E+09,9E+09,9E+09,9E+09]];
	CONST jointtarget Target_027:=[[164.374588252,-27.5,-86.25,0,30,0],[9E+09,9E+09,9E+09,9E+09,9E+09,9E+09]];
	CONST jointtarget Target_029:=[[-170,10,-148.75,0,30,0],[9E+09,9E+09,9E+09,9E+09,9E+09,9E+09]];
	CONST jointtarget Target_028:=[[-170,10,-148.75,0,30,0],[9E+09,9E+09,9E+09,9E+09,9E+09,9E+09]];
	CONST jointtarget Target_030:=[[164.374588252,10,-148.75,0,30,0],[9E+09,9E+09,9E+09,9E+09,9E+09,9E+09]];
	CONST jointtarget Target_032:=[[-168.634045402,-65,-23.75,0,30,0],[9E+09,9E+09,9E+09,9E+09,9E+09,9E+09]];
	CONST jointtarget Target_031:=[[-139.090909091,-65,-23.75,0,30,0],[9E+09,9E+09,9E+09,9E+09,9E+09,9E+09]];
	CONST jointtarget Target_033:=[[163.054803185,-65,-23.75,0,30,0],[9E+09,9E+09,9E+09,9E+09,9E+09,9E+09]];
	CONST jointtarget Target_035:=[[-168.634045402,47.5,-180,0,30,0],[9E+09,9E+09,9E+09,9E+09,9E+09,9E+09]];
	CONST jointtarget Target_034:=[[-139.090909091,47.5,-180,0,30,0],[9E+09,9E+09,9E+09,9E+09,9E+09,9E+09]];
	CONST jointtarget Target_036:=[[-167.738798847,47.5,-180,0,30,0],[9E+09,9E+09,9E+09,9E+09,9E+09,9E+09]];
	CONST jointtarget Target_038:=[[-167.268090805,10,-117.5,0,30,0],[9E+09,9E+09,9E+09,9E+09,9E+09,9E+09]];
	CONST jointtarget Target_037:=[[-108.181818182,10,-117.5,0,30,0],[9E+09,9E+09,9E+09,9E+09,9E+09,9E+09]];
	CONST jointtarget Target_039:=[[-169.058583914,10,-117.5,0,30,0],[9E+09,9E+09,9E+09,9E+09,9E+09,9E+09]];
	CONST jointtarget Target_041:=[[-167.268090805,47.5,-180,0,30,0],[9E+09,9E+09,9E+09,9E+09,9E+09,9E+09]];
	CONST jointtarget Target_040:=[[-108.181818182,47.5,-180,0,30,0],[9E+09,9E+09,9E+09,9E+09,9E+09,9E+09]];
	CONST jointtarget Target_042:=[[-169.058583914,47.5,-180,0,30,0],[9E+09,9E+09,9E+09,9E+09,9E+09,9E+09]];
	CONST jointtarget Target_044:=[[167.57720549,10,-117.5,0,30,0],[9E+09,9E+09,9E+09,9E+09,9E+09,9E+09]];
	CONST jointtarget Target_043:=[[-77.272727273,10,-117.5,0,30,0],[9E+09,9E+09,9E+09,9E+09,9E+09,9E+09]];
	CONST jointtarget Target_045:=[[-162.321149987,10,-117.5,0,30,0],[9E+09,9E+09,9E+09,9E+09,9E+09,9E+09]];
	CONST jointtarget Target_047:=[[167.57720549,47.5,-180,0,30,0],[9E+09,9E+09,9E+09,9E+09,9E+09,9E+09]];
	CONST jointtarget Target_046:=[[-77.272727273,47.5,-180,0,30,0],[9E+09,9E+09,9E+09,9E+09,9E+09,9E+09]];
	CONST jointtarget Target_048:=[[-162.321149987,47.5,-180,0,30,0],[9E+09,9E+09,9E+09,9E+09,9E+09,9E+09]];
	CONST jointtarget Target_050:=[[162.228810926,-65,-23.75,0,30,0],[9E+09,9E+09,9E+09,9E+09,9E+09,9E+09]];
	CONST jointtarget Target_049:=[[-46.363636364,-65,-23.75,0,30,0],[9E+09,9E+09,9E+09,9E+09,9E+09,9E+09]];
	CONST jointtarget Target_051:=[[-163.640935054,-65,-23.75,0,30,0],[9E+09,9E+09,9E+09,9E+09,9E+09,9E+09]];
	CONST jointtarget Target_053:=[[162.228810926,47.5,-180,0,30,0],[9E+09,9E+09,9E+09,9E+09,9E+09,9E+09]];
	CONST jointtarget Target_052:=[[-46.363636364,47.5,-180,0,30,0],[9E+09,9E+09,9E+09,9E+09,9E+09,9E+09]];
	CONST jointtarget Target_054:=[[-163.640935054,47.5,-180,0,30,0],[9E+09,9E+09,9E+09,9E+09,9E+09,9E+09]];
	CONST jointtarget Target_056:=[[158.223286194,-65,-55,0,30,0],[9E+09,9E+09,9E+09,9E+09,9E+09,9E+09]];
	CONST jointtarget Target_055:=[[-15.454545455,-65,-55,0,30,0],[9E+09,9E+09,9E+09,9E+09,9E+09,9E+09]];
	CONST jointtarget Target_057:=[[-156.903501127,-65,-55,0,30,0],[9E+09,9E+09,9E+09,9E+09,9E+09,9E+09]];
	CONST jointtarget Target_059:=[[158.223286194,-65,-23.75,0,30,0],[9E+09,9E+09,9E+09,9E+09,9E+09,9E+09]];
	CONST jointtarget Target_058:=[[-15.454545455,-65,-23.75,0,30,0],[9E+09,9E+09,9E+09,9E+09,9E+09,9E+09]];
	CONST jointtarget Target_060:=[[-156.903501127,-65,-23.75,0,30,0],[9E+09,9E+09,9E+09,9E+09,9E+09,9E+09]];
	CONST jointtarget Target_062:=[[158.223286194,-27.5,-86.25,0,30,0],[9E+09,9E+09,9E+09,9E+09,9E+09,9E+09]];
	CONST jointtarget Target_061:=[[-15.454545455,-27.5,-86.25,0,30,0],[9E+09,9E+09,9E+09,9E+09,9E+09,9E+09]];
	CONST jointtarget Target_063:=[[-156.903501127,-27.5,-86.25,0,30,0],[9E+09,9E+09,9E+09,9E+09,9E+09,9E+09]];
	CONST jointtarget Target_065:=[[158.223286194,10,-148.75,0,30,0],[9E+09,9E+09,9E+09,9E+09,9E+09,9E+09]];
	CONST jointtarget Target_064:=[[-15.454545455,10,-148.75,0,30,0],[9E+09,9E+09,9E+09,9E+09,9E+09,9E+09]];
	CONST jointtarget Target_066:=[[-156.903501127,10,-148.75,0,30,0],[9E+09,9E+09,9E+09,9E+09,9E+09,9E+09]];
	CONST jointtarget Target_068:=[[-159.118532749,-65,70,0,30,0],[9E+09,9E+09,9E+09,9E+09,9E+09,9E+09]];
	CONST jointtarget Target_067:=[[15.454545455,-65,70,0,30,0],[9E+09,9E+09,9E+09,9E+09,9E+09,9E+09]];
	CONST jointtarget Target_069:=[[169.436952896,-65,70,0,30,0],[9E+09,9E+09,9E+09,9E+09,9E+09,9E+09]];
	CONST jointtarget Target_071:=[[-159.118532749,-27.5,7.5,0,30,0],[9E+09,9E+09,9E+09,9E+09,9E+09,9E+09]];
	CONST jointtarget Target_070:=[[15.454545455,-27.5,7.5,0,30,0],[9E+09,9E+09,9E+09,9E+09,9E+09,9E+09]];
	CONST jointtarget Target_072:=[[169.436952896,-27.5,7.5,0,30,0],[9E+09,9E+09,9E+09,9E+09,9E+09,9E+09]];
	CONST jointtarget Target_074:=[[-159.118532749,-27.5,38.75,0,30,0],[9E+09,9E+09,9E+09,9E+09,9E+09,9E+09]];
	CONST jointtarget Target_073:=[[15.454545455,-27.5,38.75,0,30,0],[9E+09,9E+09,9E+09,9E+09,9E+09,9E+09]];
	CONST jointtarget Target_075:=[[169.436952896,-27.5,38.75,0,30,0],[9E+09,9E+09,9E+09,9E+09,9E+09,9E+09]];
	CONST jointtarget Target_077:=[[-159.118532749,-27.5,70,0,30,0],[9E+09,9E+09,9E+09,9E+09,9E+09,9E+09]];
	CONST jointtarget Target_076:=[[15.454545455,-27.5,70,0,30,0],[9E+09,9E+09,9E+09,9E+09,9E+09,9E+09]];
	CONST jointtarget Target_078:=[[169.436952896,-27.5,70,0,30,0],[9E+09,9E+09,9E+09,9E+09,9E+09,9E+09]];
	CONST jointtarget Target_080:=[[227.295779513,-65,70,0,30,0],[9E+09,9E+09,9E+09,9E+09,9E+09,9E+09]];
	CONST jointtarget Target_079:=[[170,-65,70,0,30,0],[9E+09,9E+09,9E+09,9E+09,9E+09,9E+09]];
	CONST jointtarget Target_081:=[[284.591559026,-65,70,0,30,0],[9E+09,9E+09,9E+09,9E+09,9E+09,9E+09]];
	CONST jointtarget Target_083:=[[227.295779513,-27.5,7.5,0,30,0],[9E+09,9E+09,9E+09,9E+09,9E+09,9E+09]];
	CONST jointtarget Target_082:=[[170,-27.5,7.5,0,30,0],[9E+09,9E+09,9E+09,9E+09,9E+09,9E+09]];
	CONST jointtarget Target_084:=[[284.591559026,-27.5,7.5,0,30,0],[9E+09,9E+09,9E+09,9E+09,9E+09,9E+09]];
	CONST jointtarget Target_086:=[[227.295779513,-27.5,38.75,0,30,0],[9E+09,9E+09,9E+09,9E+09,9E+09,9E+09]];
	CONST jointtarget Target_085:=[[170,-27.5,38.75,0,30,0],[9E+09,9E+09,9E+09,9E+09,9E+09,9E+09]];
	CONST jointtarget Target_087:=[[284.591559026,-27.5,38.75,0,30,0],[9E+09,9E+09,9E+09,9E+09,9E+09,9E+09]];
	CONST jointtarget Target_089:=[[227.295779513,-27.5,70,0,30,0],[9E+09,9E+09,9E+09,9E+09,9E+09,9E+09]];
	CONST jointtarget Target_088:=[[170,-27.5,70,0,30,0],[9E+09,9E+09,9E+09,9E+09,9E+09,9E+09]];
	CONST jointtarget Target_090:=[[284.591559026,-27.5,70,0,30,0],[9E+09,9E+09,9E+09,9E+09,9E+09,9E+09]];
	CONST jointtarget Target_092:=[[227.295779513,10,-55,0,30,0],[9E+09,9E+09,9E+09,9E+09,9E+09,9E+09]];
	CONST jointtarget Target_091:=[[170,10,-55,0,30,0],[9E+09,9E+09,9E+09,9E+09,9E+09,9E+09]];
	CONST jointtarget Target_093:=[[284.591559026,10,-55,0,30,0],[9E+09,9E+09,9E+09,9E+09,9E+09,9E+09]];
	CONST jointtarget Target_095:=[[227.295779513,10,-23.75,0,30,0],[9E+09,9E+09,9E+09,9E+09,9E+09,9E+09]];
	CONST jointtarget Target_094:=[[170,10,-23.75,0,30,0],[9E+09,9E+09,9E+09,9E+09,9E+09,9E+09]];
	CONST jointtarget Target_096:=[[284.591559026,10,-23.75,0,30,0],[9E+09,9E+09,9E+09,9E+09,9E+09,9E+09]];
	CONST jointtarget Target_098:=[[227.295779513,10,7.5,0,30,0],[9E+09,9E+09,9E+09,9E+09,9E+09,9E+09]];
	CONST jointtarget Target_097:=[[170,10,7.5,0,30,0],[9E+09,9E+09,9E+09,9E+09,9E+09,9E+09]];
	CONST jointtarget Target_099:=[[284.591559026,10,7.5,0,30,0],[9E+09,9E+09,9E+09,9E+09,9E+09,9E+09]];
	CONST jointtarget Target_0101:=[[227.295779513,10,38.75,0,30,0],[9E+09,9E+09,9E+09,9E+09,9E+09,9E+09]];
	CONST jointtarget Target_0100:=[[170,10,38.75,0,30,0],[9E+09,9E+09,9E+09,9E+09,9E+09,9E+09]];
	CONST jointtarget Target_0102:=[[284.591559026,10,38.75,0,30,0],[9E+09,9E+09,9E+09,9E+09,9E+09,9E+09]];
	CONST jointtarget Target_0104:=[[227.295779513,47.5,-117.5,0,30,0],[9E+09,9E+09,9E+09,9E+09,9E+09,9E+09]];
	CONST jointtarget Target_0103:=[[170,47.5,-117.5,0,30,0],[9E+09,9E+09,9E+09,9E+09,9E+09,9E+09]];
	CONST jointtarget Target_0105:=[[284.591559026,47.5,-117.5,0,30,0],[9E+09,9E+09,9E+09,9E+09,9E+09,9E+09]];
	CONST jointtarget Target_0107:=[[227.295779513,47.5,-86.25,0,30,0],[9E+09,9E+09,9E+09,9E+09,9E+09,9E+09]];
	CONST jointtarget Target_0106:=[[170,47.5,-86.25,0,30,0],[9E+09,9E+09,9E+09,9E+09,9E+09,9E+09]];
	CONST jointtarget Target_0108:=[[284.591559026,47.5,-86.25,0,30,0],[9E+09,9E+09,9E+09,9E+09,9E+09,9E+09]];
	CONST jointtarget Target_0110:=[[227.295779513,85,-148.75,0,30,0],[9E+09,9E+09,9E+09,9E+09,9E+09,9E+09]];
	CONST jointtarget Target_0109:=[[170,85,-148.75,0,30,0],[9E+09,9E+09,9E+09,9E+09,9E+09,9E+09]];
	CONST jointtarget Target_0111:=[[284.591559026,85,-148.75,0,30,0],[9E+09,9E+09,9E+09,9E+09,9E+09,9E+09]];

	PROC Path_10()
	    MoveJ Target_10,v3000,z100,MyNewTool\WObj:=wobj0;
	    MoveJ Target_20,v3000,z100,MyNewTool\WObj:=wobj0;
	    MoveJ Target_30,v3000,z100,MyNewTool\WObj:=wobj0;
	    MoveJ Target_40,v3000,z100,MyNewTool\WObj:=wobj0;
	    MoveJ Target_50,v3000,z100,MyNewTool\WObj:=wobj0;
		MoveJ Target_60,v3000,z100,MyNewTool\WObj:=wobj0;
		MoveJ Target_70,v3000,z100,MyNewTool\WObj:=wobj0;
		MoveJ Target_80,v3000,z100,MyNewTool\WObj:=wobj0;
		MoveAbsJ JointTarget_1,v3000,z200,MyNewTool\WObj:=wobj0;
		MoveAbsJ JointTarget_2,v3000,z200,MyNewTool\WObj:=wobj0;
		MoveAbsJ JointTarget_3,v3000,z200,MyNewTool\WObj:=wobj0;
		MoveAbsJ JointTarget_4,v3000,z200,MyNewTool\WObj:=wobj0;
		MoveAbsJ JointTarget_5,v3000,z200,MyNewTool\WObj:=wobj0;
		MoveAbsJ JointTarget_6,v3000,z200,MyNewTool\WObj:=wobj0;
		MoveAbsJ JointTarget_7,v3000,z200,MyNewTool\WObj:=wobj0;
		MoveAbsJ JointTarget_8,v3000,z200,MyNewTool\WObj:=wobj0;
		MoveAbsJ JointTarget_9,v3000,z200,MyNewTool\WObj:=wobj0;
		MoveAbsJ JointTarget_10,v3000,z200,MyNewTool\WObj:=wobj0;
		MoveAbsJ JointTarget_11,v3000,z200,MyNewTool\WObj:=wobj0;
	ENDPROC
	PROC collision0path()
	    MoveAbsJ Target_02,[6000, 5000, 5000, 5000],z100,MyNewTool\WObj:=wobj0;
	    MoveAbsJ Target_01,[6000, 5000, 5000, 5000],z100,MyNewTool\WObj:=wobj0;
		MoveAbsJ Target_03,[6000, 5000, 5000, 5000],z100,MyNewTool\WObj:=wobj0;
	ENDPROC
	PROC collision1path()
	    MoveAbsJ Target_05,[6000, 5000, 5000, 5000],z100,MyNewTool\WObj:=wobj0;
	    MoveAbsJ Target_04,[6000, 5000, 5000, 5000],z100,MyNewTool\WObj:=wobj0;
	    MoveAbsJ Target_06,[6000, 5000, 5000, 5000],z100,MyNewTool\WObj:=wobj0;
	ENDPROC
	PROC collision2path()
	    MoveAbsJ Target_08,v2000,z100,tool0\WObj:=wobj0;
	    MoveAbsJ Target_07,v2000,z100,tool0\WObj:=wobj0;
	    MoveAbsJ Target_09,v2000,z100,tool0\WObj:=wobj0;
	ENDPROC
	PROC collision3path()
	    MoveAbsJ Target_011,v1000,z100,MyNewTool\WObj:=wobj0;
	    MoveAbsJ Target_010,v1000,z100,MyNewTool\WObj:=wobj0;
	    MoveAbsJ Target_012,v1000,z100,MyNewTool\WObj:=wobj0;
	ENDPROC
	PROC collision4path()
	    MoveAbsJ Target_014,[6000, 5000, 5000, 5000],z100,MyNewTool\WObj:=wobj0;
	    MoveAbsJ Target_013,[6000, 5000, 5000, 5000],z100,MyNewTool\WObj:=wobj0;
	    MoveAbsJ Target_015,[6000, 5000, 5000, 5000],z100,MyNewTool\WObj:=wobj0;
	ENDPROC
	PROC collision5path()
	    MoveAbsJ Target_017,[6000, 5000, 5000, 5000],z100,MyNewTool\WObj:=wobj0;
	    MoveAbsJ Target_016,[6000, 5000, 5000, 5000],z100,MyNewTool\WObj:=wobj0;
		MoveAbsJ Target_018,[6000, 5000, 5000, 5000],z100,MyNewTool\WObj:=wobj0;
	ENDPROC
	PROC collision6path()
	    MoveAbsJ Target_020,[6000, 5000, 5000, 5000],z100,MyNewTool\WObj:=wobj0;
	    MoveAbsJ Target_019,[6000, 5000, 5000, 5000],z100,MyNewTool\WObj:=wobj0;
		MoveAbsJ Target_021,[6000, 5000, 5000, 5000],z100,MyNewTool\WObj:=wobj0;
	ENDPROC
	PROC collision7path()
	    MoveAbsJ Target_023,[6000, 5000, 5000, 5000],z100,MyNewTool\WObj:=wobj0;
	    MoveAbsJ Target_022,[6000, 5000, 5000, 5000],z100,MyNewTool\WObj:=wobj0;
		MoveAbsJ Target_024,[6000, 5000, 5000, 5000],z100,MyNewTool\WObj:=wobj0;
	ENDPROC
	PROC collision8path()
	    MoveAbsJ Target_026,[6000, 5000, 5000, 5000],z100,MyNewTool\WObj:=wobj0;
	    MoveAbsJ Target_025,[6000, 5000, 5000, 5000],z100,MyNewTool\WObj:=wobj0;
	    MoveAbsJ Target_027,[6000, 5000, 5000, 5000],z100,MyNewTool\WObj:=wobj0;
	ENDPROC
	PROC collision9path()
	    MoveAbsJ Target_029,[6000, 5000, 5000, 5000],z100,MyNewTool\WObj:=wobj0;
	    MoveAbsJ Target_028,[6000, 5000, 5000, 5000],z100,MyNewTool\WObj:=wobj0;
		MoveAbsJ Target_030,[6000, 5000, 5000, 5000],z100,MyNewTool\WObj:=wobj0;
	ENDPROC
	PROC collision10path()
	    MoveAbsJ Target_032,[6000, 5000, 5000, 5000],z100,MyNewTool\WObj:=wobj0;
	    MoveAbsJ Target_031,[6000, 5000, 5000, 5000],z100,MyNewTool\WObj:=wobj0;
	    MoveAbsJ Target_033,[6000, 5000, 5000, 5000],z100,MyNewTool\WObj:=wobj0;
	ENDPROC
	PROC collision11path()
	    MoveAbsJ Target_035,[6000, 5000, 5000, 5000],z100,MyNewTool\WObj:=wobj0;
	    MoveAbsJ Target_034,[6000, 5000, 5000, 5000],z100,MyNewTool\WObj:=wobj0;
	    MoveAbsJ Target_036,[6000, 5000, 5000, 5000],z100,MyNewTool\WObj:=wobj0;
	ENDPROC
	PROC collision12path()
	    MoveAbsJ Target_038,[6000, 5000, 5000, 5000],z100,MyNewTool\WObj:=wobj0;
	    MoveAbsJ Target_037,[6000, 5000, 5000, 5000],z100,MyNewTool\WObj:=wobj0;
	    MoveAbsJ Target_039,[6000, 5000, 5000, 5000],z100,MyNewTool\WObj:=wobj0;
	ENDPROC
	PROC collision13path()
	    MoveAbsJ Target_041,[6000, 5000, 5000, 5000],z100,MyNewTool\WObj:=wobj0;
	    MoveAbsJ Target_040,[6000, 5000, 5000, 5000],z100,MyNewTool\WObj:=wobj0;
	    MoveAbsJ Target_042,[6000, 5000, 5000, 5000],z100,MyNewTool\WObj:=wobj0;
	ENDPROC
	PROC collision14path()
	    MoveAbsJ Target_044,[6000, 5000, 5000, 5000],z100,MyNewTool\WObj:=wobj0;
	    MoveAbsJ Target_043,[6000, 5000, 5000, 5000],z100,MyNewTool\WObj:=wobj0;
	    MoveAbsJ Target_045,[6000, 5000, 5000, 5000],z100,MyNewTool\WObj:=wobj0;
	ENDPROC
	PROC collision15path()
	    MoveAbsJ Target_047,[6000, 5000, 5000, 5000],z100,MyNewTool\WObj:=wobj0;
	    MoveAbsJ Target_046,[6000, 5000, 5000, 5000],z100,MyNewTool\WObj:=wobj0;
	    MoveAbsJ Target_048,[6000, 5000, 5000, 5000],z100,MyNewTool\WObj:=wobj0;
	ENDPROC
	PROC collision16path()
	    MoveAbsJ Target_050,[6000, 5000, 5000, 5000],z100,MyNewTool\WObj:=wobj0;
	    MoveAbsJ Target_049,[6000, 5000, 5000, 5000],z100,MyNewTool\WObj:=wobj0;
	    MoveAbsJ Target_051,[6000, 5000, 5000, 5000],z100,MyNewTool\WObj:=wobj0;
	ENDPROC
	PROC collision17path()
	    MoveAbsJ Target_053,[6000, 5000, 5000, 5000],z100,MyNewTool\WObj:=wobj0;
	    MoveAbsJ Target_052,[6000, 5000, 5000, 5000],z100,MyNewTool\WObj:=wobj0;
	    MoveAbsJ Target_054,[6000, 5000, 5000, 5000],z100,MyNewTool\WObj:=wobj0;
	ENDPROC
	PROC collision18path()
	    MoveAbsJ Target_056,[6000, 5000, 5000, 5000],z100,MyNewTool\WObj:=wobj0;
	    MoveAbsJ Target_055,[6000, 5000, 5000, 5000],z100,MyNewTool\WObj:=wobj0;
	    MoveAbsJ Target_057,[6000, 5000, 5000, 5000],z100,MyNewTool\WObj:=wobj0;
	ENDPROC
	PROC collision19path()
	    MoveAbsJ Target_059,[6000, 5000, 5000, 5000],z100,MyNewTool\WObj:=wobj0;
	    MoveAbsJ Target_058,[6000, 5000, 5000, 5000],z100,MyNewTool\WObj:=wobj0;
	    MoveAbsJ Target_060,[6000, 5000, 5000, 5000],z100,MyNewTool\WObj:=wobj0;
	ENDPROC
	PROC collision20path()
	    MoveAbsJ Target_062,[6000, 5000, 5000, 5000],z100,MyNewTool\WObj:=wobj0;
	    MoveAbsJ Target_061,[6000, 5000, 5000, 5000],z100,MyNewTool\WObj:=wobj0;
	    MoveAbsJ Target_063,[6000, 5000, 5000, 5000],z100,MyNewTool\WObj:=wobj0;
	ENDPROC
	PROC collision21path()
	    MoveAbsJ Target_065,[6000, 5000, 5000, 5000],z100,MyNewTool\WObj:=wobj0;
	    MoveAbsJ Target_064,[6000, 5000, 5000, 5000],z100,MyNewTool\WObj:=wobj0;
	    MoveAbsJ Target_066,[6000, 5000, 5000, 5000],z100,MyNewTool\WObj:=wobj0;
	ENDPROC
	PROC collision22path()
	    MoveAbsJ Target_068,[6000, 5000, 5000, 5000],z100,MyNewTool\WObj:=wobj0;
	    MoveAbsJ Target_067,[6000, 5000, 5000, 5000],z100,MyNewTool\WObj:=wobj0;
	    MoveAbsJ Target_069,[6000, 5000, 5000, 5000],z100,MyNewTool\WObj:=wobj0;
	ENDPROC
	PROC collision23path()
	    MoveAbsJ Target_071,[6000, 5000, 5000, 5000],z100,MyNewTool\WObj:=wobj0;
	    MoveAbsJ Target_070,[6000, 5000, 5000, 5000],z100,MyNewTool\WObj:=wobj0;
	    MoveAbsJ Target_072,[6000, 5000, 5000, 5000],z100,MyNewTool\WObj:=wobj0;
	ENDPROC
	PROC collision24path()
	    MoveAbsJ Target_074,[6000, 5000, 5000, 5000],z100,MyNewTool\WObj:=wobj0;
	    MoveAbsJ Target_073,[6000, 5000, 5000, 5000],z100,MyNewTool\WObj:=wobj0;
	    MoveAbsJ Target_075,[6000, 5000, 5000, 5000],z100,MyNewTool\WObj:=wobj0;
	ENDPROC
	PROC collision25path()
	    MoveAbsJ Target_077,[6000, 5000, 5000, 5000],z100,MyNewTool\WObj:=wobj0;
	    MoveAbsJ Target_076,[6000, 5000, 5000, 5000],z100,MyNewTool\WObj:=wobj0;
	    MoveAbsJ Target_078,[6000, 5000, 5000, 5000],z100,MyNewTool\WObj:=wobj0;
	ENDPROC
	PROC collision26path()
	    MoveAbsJ Target_080,[6000, 5000, 5000, 5000],z100,MyNewTool\WObj:=wobj0;
	    MoveAbsJ Target_079,[6000, 5000, 5000, 5000],z100,MyNewTool\WObj:=wobj0;
	    MoveAbsJ Target_081,[6000, 5000, 5000, 5000],z100,MyNewTool\WObj:=wobj0;
	ENDPROC
	PROC collision27path()
	    MoveAbsJ Target_083,[6000, 5000, 5000, 5000],z100,MyNewTool\WObj:=wobj0;
	    MoveAbsJ Target_082,[6000, 5000, 5000, 5000],z100,MyNewTool\WObj:=wobj0;
	    MoveAbsJ Target_084,[6000, 5000, 5000, 5000],z100,MyNewTool\WObj:=wobj0;
	ENDPROC
	PROC collision28path()
	    MoveAbsJ Target_086,[6000, 5000, 5000, 5000],z100,MyNewTool\WObj:=wobj0;
	    MoveAbsJ Target_085,[6000, 5000, 5000, 5000],z100,MyNewTool\WObj:=wobj0;
	    MoveAbsJ Target_087,[6000, 5000, 5000, 5000],z100,MyNewTool\WObj:=wobj0;
	ENDPROC
	PROC collision29path()
	    MoveAbsJ Target_089,[6000, 5000, 5000, 5000],z100,MyNewTool\WObj:=wobj0;
	    MoveAbsJ Target_088,[6000, 5000, 5000, 5000],z100,MyNewTool\WObj:=wobj0;
	    MoveAbsJ Target_090,[6000, 5000, 5000, 5000],z100,MyNewTool\WObj:=wobj0;
	ENDPROC
	PROC collision30path()
	    MoveAbsJ Target_092,[6000, 5000, 5000, 5000],z100,MyNewTool\WObj:=wobj0;
	    MoveAbsJ Target_091,[6000, 5000, 5000, 5000],z100,MyNewTool\WObj:=wobj0;
	    MoveAbsJ Target_093,[6000, 5000, 5000, 5000],z100,MyNewTool\WObj:=wobj0;
	ENDPROC
	PROC collision31path()
	    MoveAbsJ Target_095,[6000, 5000, 5000, 5000],z100,MyNewTool\WObj:=wobj0;
	    MoveAbsJ Target_094,[6000, 5000, 5000, 5000],z100,MyNewTool\WObj:=wobj0;
	    MoveAbsJ Target_096,[6000, 5000, 5000, 5000],z100,MyNewTool\WObj:=wobj0;
	ENDPROC
	PROC collision32path()
	    MoveAbsJ Target_098,[6000, 5000, 5000, 5000],z100,MyNewTool\WObj:=wobj0;
	    MoveAbsJ Target_097,[6000, 5000, 5000, 5000],z100,MyNewTool\WObj:=wobj0;
	    MoveAbsJ Target_099,[6000, 5000, 5000, 5000],z100,MyNewTool\WObj:=wobj0;
	ENDPROC
	PROC collision33path()
	    MoveAbsJ Target_0101,[6000, 5000, 5000, 5000],z100,MyNewTool\WObj:=wobj0;
	    MoveAbsJ Target_0100,[6000, 5000, 5000, 5000],z100,MyNewTool\WObj:=wobj0;
	    MoveAbsJ Target_0102,[6000, 5000, 5000, 5000],z100,MyNewTool\WObj:=wobj0;
	ENDPROC
	PROC collision34path()
	    MoveAbsJ Target_0104,[6000, 5000, 5000, 5000],z100,MyNewTool\WObj:=wobj0;
	    MoveAbsJ Target_0103,[6000, 5000, 5000, 5000],z100,MyNewTool\WObj:=wobj0;
	    MoveAbsJ Target_0105,[6000, 5000, 5000, 5000],z100,MyNewTool\WObj:=wobj0;
	ENDPROC
	PROC collision35path()
	    MoveAbsJ Target_0107,[6000, 5000, 5000, 5000],z100,MyNewTool\WObj:=wobj0;
	    MoveAbsJ Target_0106,[6000, 5000, 5000, 5000],z100,MyNewTool\WObj:=wobj0;
	    MoveAbsJ Target_0108,[6000, 5000, 5000, 5000],z100,MyNewTool\WObj:=wobj0;
	ENDPROC
	PROC collision36path()
	    MoveAbsJ Target_0110,[6000, 5000, 5000, 5000],z100,MyNewTool\WObj:=wobj0;
	    MoveAbsJ Target_0109,[6000, 5000, 5000, 5000],z100,MyNewTool\WObj:=wobj0;
	    MoveAbsJ Target_0111,[6000, 5000, 5000, 5000],z100,MyNewTool\WObj:=wobj0;
	ENDPROC

ENDMODULE

--- Backups/IRB_6700_175kg_3.05m/RAPID/TASK1/SYSMOD/LINKEDM.sys ---
%%%
  VERSION:1
  LANGUAGE:ENGLISH
%%%

MODULE LINKEDM (SYSMODULE)

! FOLLOWER
!     Name of electronically linked follower axis used by operator at teach pendent.
      PERS string l_f_axis_name{5}       :=  ["",  "", "", "", ""];

!     Name of the mechanical unit for follower axis.
      PERS string l_f_mecunt_n{5}  :=  ["", "", "", "", ""];

!     Linked follower axis number in the mechanical unit (first axis in mech. unit is number 1).
      PERS num l_f_axis_no{5}      :=  [0,          0,   0,  0,  0];

! MASTER
!     Name of the mechanical unit for linked master axis.
      PERS string l_m_mecunt_n{5} :=  ["", "", "", "", ""];

!     Linked master axis number in the mechanical unit (first axis in mech. unit is number 1).
!     See axis number table in documentation for different master mechanical units.
      PERS num l_m_axis_no{5}     :=  [0,  0,  0,  0,  0];

! POSITION OFFSET
!     The increase of the allowed offset position between the master and follower
!     positions, used when starting AUTO mode. As soon as the offset is decreased
!     the old configurated parameter is used.
!     Example: 3 => the configurated value of allowed offset is increased 3 times.
      PERS num offset_ratio{5}       :=  [10,  10,   10,  10,  10];

! SPEED RATIO
!     Speed_ratio used in AUTO and JOG modes [ very_slow   slow    normal    fast]
!     Value 1 = max allowed manual speed.
      CONST num speed_ratio {20}      := [0.01, 0.01, 0.01, 0.01, 0.01,
                                          0.05, 0.05, 0.05, 0.05, 0.05,
                                          0.20, 0.20, 0.20, 0.20, 0.20,
                                          1.00, 1.00, 1.00, 1.00, 1.00];

! STEP SIZE
!     Displacement position used in JOG mode for each activation of positive or
!     negative movement.                  [very_short    short   normal   long]
!     Unit degees or meter.
      CONST num displacement {20}     := [0.001, 0.001, 0.001, 0.001, 0.001,
                                          0.005, 0.005, 0.005, 0.005, 0.005,
                                          0.020, 0.020, 0.020, 0.020, 0.020,
                                          0.100, 0.100, 0.100, 0.100, 0.100];


!-------------------------------------------------------------
 PROC Linked_m ()
      Linked_m_exe ;
 ENDPROC
ENDMODULE
